ABB RAPID module: SERVER.mod

MODULE SERVER
!
!  Released under MIT License
!
!  David Pollard
!  Bristol Robotics Laboratory
!
!  Original author
!  Michael Dawson-Haggerty
!
!

!////////////////
!GLOBAL VARIABLES
!////////////////

! Robot configuration
PERS tooldata currentTool := [TRUE,[[-44.5,9.9,114],[1,0,0,0]],[0.001,[0,0,0.001],[1,0,0,0],0,0,0]];
PERS wobjdata currentWobj := [FALSE,TRUE,"",[[0,0,0],[1,0,0,0]],[[633.5,9.9,380],[1,0,0,0]]];
PERS speeddata currentSpeed;
PERS zonedata currentZone;

! Clock Synchronization
PERS bool startLog:=TRUE;
PERS bool startRob:=TRUE;

! Mutex between logger and changing the tool and work objects
PERS bool frameMutex:=FALSE;

! PC communication
VAR socketdev clientSocket;
VAR socketdev serverSocket;
VAR num instructionCode;
VAR num params{10};
VAR num nParams;

VAR num qOrientation{4};  !store Q value for orientation
VAR num tempNum;          !For use whenever needed. Don't rely on it to stay the same

!PERS string ipController:= "192.168.125.1"; !robot default IP
PERS string ipController:= "127.0.0.1"; !local IP for testing in simulation
PERS num serverPort:= 5000;

! Motion of the robot
VAR robtarget cartesianTarget;
VAR jointtarget jointsTarget;
VAR bool moveCompleted; !Set to true after finishing a Move instruction.

! Buffered move variables
CONST num MAX_BUFFER := 512;
CONST num MAX_SAVED_BUFFERS := 20;
VAR num BUFFER_POS := 0;
VAR robtarget bufferTargets{MAX_BUFFER};
VAR speeddata bufferSpeeds{MAX_BUFFER};
VAR bool extrudeDuringBufferMove;

! Spare buffers for saving paths
VAR robtarget savedBufferTargets{MAX_SAVED_BUFFERS, MAX_BUFFER};
VAR speeddata savedBufferSpeeds{MAX_SAVED_BUFFERS, MAX_BUFFER};
VAR num savedBufferPos{MAX_SAVED_BUFFERS};

! External axis position variables
VAR extjoint externalAxis;

! Circular move buffer
VAR robtarget circPoint;

! Correct Instruction Execution and possible return values
VAR num ok;
CONST num SERVER_BAD_MSG :=  0;
CONST num SERVER_OK := 1;
TASK PERS tooldata testNozzle:=[TRUE,[[-47.7913,12.961,103.954],[1,0,0,0]],[0.5,[0,0,0],[1,0,0,0],0,0,0]];
TASK PERS tooldata nozzle:=[TRUE,[[-44.5058,10.7853,113.761],[1,0,0,0]],[1,[0,0,0],[1,0,0,0],0,0,0]];


!////////////////
!LOCAL METHODS
!////////////////

! Method to parse the message received from a PC
!  If correct message, loads values on:
!  - instructionCode.
!  - nParams: Number of received parameters.
!  - params{nParams}: Vector of received params.
PROC ParseMsg(string msg)
    !//Local variables
    VAR bool auxOk;
    VAR num ind:=1;
    VAR num newInd;
    VAR num length;
    VAR num indParam:=1;
    VAR string subString;
    VAR bool end := FALSE;

    ! Find the end character
    length := StrMatch(msg,1,"#");
    IF length > StrLen(msg) THEN
        ! Corrupt message
        nParams := -1;
    ELSE
        ! Read Instruction code
        newInd := StrMatch(msg,ind," ") + 1;
        subString := StrPart(msg,ind,newInd - ind - 1);
        auxOk:= StrToVal(subString, instructionCode);
        IF auxOk = FALSE THEN
            ! Impossible to read instruction code
            nParams := -1;
        ELSE
            ind := newInd;
            ! Read all instruction parameters (maximum of 8)
            WHILE end = FALSE DO
                newInd := StrMatch(msg,ind," ") + 1;
                IF newInd > length THEN
                    end := TRUE;
                ELSE
                    subString := StrPart(msg,ind,newInd - ind - 1);
                    auxOk := StrToVal(subString, params{indParam});
                    indParam := indParam + 1;
                    ind := newInd;
                ENDIF
            ENDWHILE
            nParams:= indParam - 1;
        ENDIF
    ENDIF
ENDPROC


! Handshake between server and client:
!  - Creates socket.
!  - Waits for incoming TCP connection.
PROC ServerCreateAndConnect(string ip, num port)
    VAR string clientIP;

    SocketCreate serverSocket;
    SocketBind serverSocket, ip, port;
    SocketListen serverSocket;
    TPWrite "SERVER: Server waiting for incoming connections ...";
    WHILE SocketGetStatus(clientSocket) <> SOCKET_CONNECTED DO
        SocketAccept serverSocket,clientSocket \ClientAddress:=clientIP \Time:=WAIT_MAX;
        IF SocketGetStatus(clientSocket) <> SOCKET_CONNECTED THEN
            TPWrite "SERVER: Problem serving an incoming connection.";
            TPWrite "SERVER: Try reconnecting.";
        ENDIF
        ! Wait 0.5 seconds for the next reconnection
        WaitTime 0.5;
    ENDWHILE
    TPWrite "SERVER: Connected to IP " + clientIP;
ENDPROC


! Parameter initialization
!  Loads default values for
!  - Tool.
!  - WorkObject.
!  - Zone.
!  - Speed.
PROC Initialize()
    currentTool := [TRUE,[[0,0,0],[1,0,0,0]],[0.001,[0,0,0.001],[1,0,0,0],0,0,0]];
    currentWobj := [FALSE,TRUE,"",[[0,0,0],[1,0,0,0]],[[0,0,0],[1,0,0,0]]];
    currentSpeed := [100, 50, 0, 0];
    currentZone := [FALSE, 0.3, 0.3,0.3,0.03,0.3,0.03]; !z0

	!Find the current external axis values so they don't move when we start
    ActUnit STN1;
	jointsTarget := CJointT();
	externalAxis := jointsTarget.extax;
ENDPROC


!////////////////////////
!//SERVER: Main procedure
!////////////////////////
PROC ServerMain()
    ! Local variables
    VAR string receivedString;   ! Received string
    VAR string sendString;       ! Reply string
    VAR string addString;        ! String to add to the reply.
    VAR bool connected;          ! Client connected
    VAR bool reconnected;        ! Drop and reconnection happened during serving a command
    VAR robtarget cartesianPose;
    VAR jointtarget jointsPose;

    ! Motion configuration
    ConfL \Off;
    SingArea \Wrist;
    moveCompleted:= TRUE;

    ! Initialization of WorkObject, Tool, Speed and Zone
    Initialize;

    ! Socket connection
    connected:=FALSE;
    ServerCreateAndConnect ipController,serverPort;
    connected:=TRUE;

    ! Server Loop
    WHILE TRUE DO
        ! Initialization of program flow variables
        ok:=SERVER_OK;              ! Correctness of executed instruction.
        reconnected:=FALSE;         ! Has communication dropped after receiving a command?
        addString := "";

        ! Wait for a command
        SocketReceive clientSocket \Str:=receivedString \Time:=WAIT_MAX;
        ParseMsg receivedString;

        ! Execution of the command
        TEST instructionCode
            CASE -1:
                IF nParams = 1 THEN
                    IF params{1} = -1 THEN
                        ChangeExtruderState (0);
                        DeactUnit STN1;
                    ELSEIF params{1} = 0 THEN
                        ResetRobotPosition;
                        ChangeExtruderState(0);
                        DeactUnit STN1;
                    ELSEIF params{1} = 1 THEN
                        ResetRobotPosition;
                        ChangeExtruderState(1);
                        ActUnit STN1;
                    ELSEIF params{1} = 2 THEN
                        ChangeExtruderState(1);
                        ActUnit STN1;
                    ENDIF
                    ok := SERVER_OK;
                ELSE
                    ok := SERVER_BAD_MSG;
                ENDIF


            CASE 0: !Ping
                IF nParams = 0 THEN
                    ok := SERVER_OK;
                ELSE
                    ok := SERVER_BAD_MSG;
                ENDIF

            CASE 1: !Cartesian Move
                IF nParams = 8 THEN
                    jointsTarget := CJointT();
	                externalAxis := jointsTarget.extax;

                    cartesianTarget :=[[params{2},params{3},params{4}],
                                       [params{5},params{6},params{7},params{8}],
                                       [0,0,0,0],
                                       externalAxis];
                    ok := SERVER_OK;
                    moveCompleted := FALSE;
                    IF params{1}=1 THEN
                        MoveL cartesianTarget, currentSpeed, fine, currentTool \WObj:=currentWobj ;
                    ELSE
                        MoveL cartesianTarget, currentSpeed, currentZone, currentTool \WObj:=currentWobj ;
                    ENDIF
                    moveCompleted := TRUE;
                ELSE
                    ok := SERVER_BAD_MSG;
                ENDIF

            CASE 2: !Joint Move
                IF nParams = 6 THEN
                    jointsTarget := CJointT();
                    externalAxis := jointsTarget.extax;

                    jointsTarget:=[[params{1},params{2},params{3},params{4},params{5},params{6}], externalAxis];
                    ok := SERVER_OK;
                    moveCompleted := FALSE;
                    MoveAbsJ jointsTarget, currentSpeed, currentZone, currentTool \Wobj:=currentWobj;
                    moveCompleted := TRUE;
                ELSE
                    ok :=SERVER_BAD_MSG;
                ENDIF

            CASE 3: !Get Cartesian Coordinates (with current tool and workobject)
                IF nParams = 0 THEN
                    cartesianPose := CRobT(\Tool:=currentTool \WObj:=currentWObj);
                    addString := NumToStr(cartesianPose.trans.x,2) + " ";
                    addString := addString + NumToStr(cartesianPose.trans.y,2) + " ";
                    addString := addString + NumToStr(cartesianPose.trans.z,2) + " ";
                    addString := addString + NumToStr(cartesianPose.rot.q1,3) + " ";
                    addString := addString + NumToStr(cartesianPose.rot.q2,3) + " ";
                    addString := addString + NumToStr(cartesianPose.rot.q3,3) + " ";
                    addString := addString + NumToStr(cartesianPose.rot.q4,3); !End of string
                    ok := SERVER_OK;
                ELSE
                    ok :=SERVER_BAD_MSG;
                ENDIF

            CASE 4: !Get Joint Coordinates
                IF nParams = 0 THEN
                    jointsPose := CJointT();
                    addString := NumToStr(jointsPose.robax.rax_1,2) + " ";
                    addString := addString + NumToStr(jointsPose.robax.rax_2,2) + " ";
                    addString := addString + NumToStr(jointsPose.robax.rax_3,2) + " ";
                    addString := addString + NumToStr(jointsPose.robax.rax_4,2) + " ";
                    addString := addString + NumToStr(jointsPose.robax.rax_5,2) + " ";
                    addString := addString + NumToStr(jointsPose.robax.rax_6,2); !End of string
                    ok := SERVER_OK;
                ELSE
                    ok:=SERVER_BAD_MSG;
                ENDIF

			CASE 5: !Get external axis positions
                IF nParams=0 THEN
                    jointsTarget:=CJointT();
                    addString:=ValToStr(jointsTarget.extax.eax_b)+" ";
                    addString:=addString + ValToStr(jointsTarget.extax.eax_c);
                    ok:=SERVER_OK;
                ELSE
                    ok:=SERVER_BAD_MSG;
                ENDIF            CASE 6: !Set Tool
                IF nParams = 7 THEN
		            WHILE (frameMutex) DO
		                WaitTime .01; !  If the frame is being used by logger, wait here
		            ENDWHILE
		            frameMutex:= TRUE;
                    currentTool.tframe.trans.x:=params{1};
                    currentTool.tframe.trans.y:=params{2};
                    currentTool.tframe.trans.z:=params{3};
                    currentTool.tframe.rot.q1:=params{4};
                    currentTool.tframe.rot.q2:=params{5};
                    currentTool.tframe.rot.q3:=params{6};
                    currentTool.tframe.rot.q4:=params{7};
                    ok := SERVER_OK;
		            frameMutex:= FALSE;
                ELSE
                    ok:=SERVER_BAD_MSG;
                ENDIF

            CASE 7: !Set Work Object
                IF nParams = 7 THEN
                    currentWobj.oframe.trans.x:=params{1};
                    currentWobj.oframe.trans.y:=params{2};
                    currentWobj.oframe.trans.z:=params{3};
                    currentWobj.oframe.rot.q1:=params{4};
                    currentWobj.oframe.rot.q2:=params{5};
                    currentWobj.oframe.rot.q3:=params{6};
                    currentWobj.oframe.rot.q4:=params{7};
                    ok := SERVER_OK;
                ELSE
                    ok:=SERVER_BAD_MSG;
                ENDIF

            CASE 8: !Set Speed of the Robot
                IF nParams = 4 THEN
                    currentSpeed.v_tcp:=params{1};
                    currentSpeed.v_ori:=params{2};
                    currentSpeed.v_leax:=params{3};
                    currentSpeed.v_reax:=params{4};
                    ok := SERVER_OK;
                ELSEIF nParams = 2 THEN
					currentSpeed.v_tcp:=params{1};
					currentSpeed.v_ori:=params{2};
					ok := SERVER_OK;
				ELSE
                    ok:=SERVER_BAD_MSG;
                ENDIF

            CASE 9: !Set zone data
                IF nParams = 4 THEN
                    IF params{1}=1 THEN
                        currentZone.finep := TRUE;
                        currentZone.pzone_tcp := 0.0;
                        currentZone.pzone_ori := 0.0;
                        currentZone.zone_ori := 0.0;
                    ELSE
                        currentZone.finep := FALSE;
                        currentZone.pzone_tcp := params{2};
                        currentZone.pzone_ori := params{3};
                        currentZone.zone_ori := params{4};
                    ENDIF
                    ok := SERVER_OK;
                ELSE
                    ok:=SERVER_BAD_MSG;
                ENDIF

            CASE 10: !Rotate about tool Z axis
                IF nParams = 1 THEN
                    ok := SERVER_OK;
                    RotateToolZ(params{1});
                ELSE
                    ok := SERVER_BAD_MSG;
                ENDIF

            CASE 11: !Check and fix Joint 6 angle
                IF nParams = 0 THEN
                    ok := SERVER_OK;
                    jointsTarget := CJointT();
                    tempNum := jointsTarget.robax.rax_6;
                    ! Move and rotate if necessary
                    IF tempNum > 270 THEN
                        TPWrite "Performing angle correction";
                        cartesianPose := CRobT();
                        MoveL RelTool(cartesianPose,0,0,-50),v100,fine,currentTool \WObj:=currentWobj;
                        RotateToolZ(-360);
                        MoveL cartesianPose,v100,fine,currentTool \WObj:=currentWobj;
                    ELSEIF tempNum < -90 THEN
                        TPWrite "Performing angle correction";
                        cartesianPose := CRobT();
                        MoveL RelTool(cartesianPose,0,0,-50),v100,fine,currentTool \WObj:=currentWobj;
                        RotateToolZ(360);
                        MoveL cartesianPose,v100,fine,currentTool \WObj:=currentWobj;
                    ENDIF
                ELSE
                    ok := SERVER_BAD_MSG;
                ENDIF


            CASE 29:
                IF nParams = 4 THEN
                    qOrientation{1} := params{1};
                    qOrientation{2} := params{2};
                    qOrientation{3} := params{3};
                    qOrientation{4} := params{4};
                    ok:=SERVER_OK;
                ELSE
                    ok:=SERVER_BAD_MSG;
                ENDIF

            CASE 30: !Add Cartesian Coordinates to buffer
                IF nParams = 7 OR nParams = 8 THEN
                    ! If external axis is necessary
                    jointsTarget := CJointT();
                    externalAxis := jointsTarget.extax;
                    IF nParams = 8 THEN
                        externalAxis.eax_c := params{8};
                    ENDIF

                    cartesianTarget :=[[params{1},params{2},params{3}],
                                        [params{4},params{5},params{6},params{7}],
                                        [0,0,0,0],
                                        externalAxis];
                    IF BUFFER_POS < MAX_BUFFER THEN
                        BUFFER_POS := BUFFER_POS + 1;
                        bufferTargets{BUFFER_POS} := cartesianTarget;
                        bufferSpeeds{BUFFER_POS} := currentSpeed;
                    ENDIF
                    ! Update Q orienatation
                    qOrientation{1} := params{4};
                    qOrientation{2} := params{5};
                    qOrientation{3} := params{6};
                    qOrientation{4} := params{7};
                    ok := SERVER_OK;
                ELSEIF nParams = 3 THEN
                    cartesianTarget :=[[params{1},params{2},params{3}],
                                        [qOrientation{1},qOrientation{2},qOrientation{3},qOrientation{4}],
                                        [0,0,0,0],
                                        externalAxis];
                    IF BUFFER_POS < MAX_BUFFER THEN
                        BUFFER_POS := BUFFER_POS + 1;
                        bufferTargets{BUFFER_POS} := cartesianTarget;
                        bufferSpeeds{BUFFER_POS} := currentSpeed;
                    ENDIF
                    ok:=SERVER_OK;
                ELSE
                    ok:=SERVER_BAD_MSG;
                ENDIF

            CASE 31: !Clear Cartesian Buffer
                IF nParams = 0 THEN
                    BUFFER_POS := 0;
                    ok := SERVER_OK;
                ELSE
                    ok:=SERVER_BAD_MSG;
                ENDIF

            CASE 32: !Get Buffer Size)
                IF nParams = 0 THEN
                    addString := NumToStr(BUFFER_POS,2);
                    ok := SERVER_OK;
                ELSE
                    ok:=SERVER_BAD_MSG;
                ENDIF

            CASE 33: !Execute moves in cartesianBuffer as linear moves NB: Circ buffer is 37
                IF nParams = 0 OR nParams = 1 THEN
                    IF nParams = 1 THEN
                        MoveL bufferTargets{1}, v100, fine, currentTool, \WObj:=currentWobj ;
                        SetDO DO10_2, 1;
                        ! Ensure signal is synchronised
                        MoveL bufferTargets{1}, v100, fine, currentTool, \WObj:=currentWobj ;
                    ENDIF

                    FOR i FROM 1 TO (BUFFER_POS) DO
                        MoveL bufferTargets{i}, bufferSpeeds{i}, currentZone, currentTool, \WObj:=currentWobj ;
                    ENDFOR

                    MoveL bufferTargets{(BUFFER_POS)}, bufferSpeeds{(BUFFER_POS)}, fine, currentTool, \WObj:=currentWobj ;

                    IF nParams = 1 THEN
                        SetDO DO10_2, 0;
                        MoveL RelTool(bufferTargets{(BUFFER_POS)},0,0,-5),v100,z1, currentTool, \WObj:=currentWobj ;
                    ENDIF


                    ok := SERVER_OK;
                ELSE
                    ok:=SERVER_BAD_MSG;
                ENDIF

            CASE 34: !External Axis move
                IF nParams = 2 THEN
                    jointsTarget := CJointT();
                    jointsTarget.extax.eax_b := params{1};
                    jointsTarget.extax.eax_c := params{2};
                    ok := SERVER_OK;
                    moveCompleted := FALSE;
                    MoveAbsJ jointsTarget, currentSpeed, fine, currentTool \Wobj:=currentWobj;
                    moveCompleted := TRUE;
                ELSE
                    ok :=SERVER_BAD_MSG;
                ENDIF

            CASE 35: !Specify circPoint for circular move, and then wait on toPoint
                IF nParams = 7 THEN
                    jointsTarget := CJointT();
                    externalAxis := jointsTarget.extax;

                    circPoint :=[[params{1},params{2},params{3}],
                                [params{4},params{5},params{6},params{7}],
                                [0,0,0,0],
                                externalAxis];
                    TPWrite "z: ", \Num:=params{3};
                    ok := SERVER_OK;
                ELSE
                    ok:=SERVER_BAD_MSG;
                ENDIF

            CASE 36: !specify toPoint, and use circPoint specified previously
                IF nParams = 7 THEN
                    jointsTarget := CJointT();
                    externalAxis := jointsTarget.extax;

                    cartesianTarget :=[[params{1},params{2},params{3}],
                                        [params{4},params{5},params{6},params{7}],
                                        [0,0,0,0],
                                        externalAxis];
                    MoveC circPoint, cartesianTarget, currentSpeed, currentZone, currentTool \WObj:=currentWobj ;
                    ok := SERVER_OK;
                ELSE
                    ok:=SERVER_BAD_MSG;
                ENDIF

            CASE 37: !execute buffer as a circular move
                IF nParams = 0 THEN
                    MoveC bufferTargets{1}, bufferTargets{2}, bufferSpeeds{1}, currentZone, currentTool \WObj:=currentWobj ;
                    ok  := SERVER_OK;
                ELSE
                    ok := SERVER_BAD_MSG;
                ENDIF


            CASE 40:  ! Find if position is reachable
                ! NB: Not recommended for calling during operation, no error handling.
                cartesianTarget :=[[params{1},params{2},params{3}],
                                    [params{4},params{5},params{6},params{7}],
                                    [0,0,0,0],
                                    externalAxis];
                IF CheckPositionReachable(cartesianTarget, currentTool, currentWobj) THEN
                    ok := SERVER_OK;
                ELSE
                    ok := SERVER_BAD_MSG;
                ENDIF




            CASE 50: !Save current buffer into existing buffer
                IF nParams = 1 THEN
                    IF params{1} < MAX_SAVED_BUFFERS THEN
                        ok := SERVER_OK;
                        TPWrite "Saved: ",\Num:=params{1};
                        FOR i FROM 1 TO BUFFER_POS DO
                            savedBufferTargets{params{1},i} := bufferTargets{i};
                            savedBufferSpeeds{params{1},i} := bufferSpeeds{i};
                        ENDFOR
                        savedBufferPos{params{1}} := BUFFER_POS;
                    ELSE
                        ErrWrite "Buffer error", "Requested buffer does not exist";
                        ok := SERVER_BAD_MSG;
                    ENDIF
                ELSE
                    ok := SERVER_BAD_MSG;
                ENDIF

            CASE 51: !Load saved buffer into current buffer. Reset BUFFER_POS
                IF nParams=1 THEN
                    IF params{1} < MAX_SAVED_BUFFERS THEN
                        ok:=SERVER_OK;
                        BUFFER_POS := savedBufferPos{params{1}};
                        FOR i FROM 1 TO BUFFER_POS DO
                            bufferTargets{i} := savedBufferTargets{params{1},i};
                            bufferSpeeds{i} := savedBufferSpeeds{params{1},i};
                        ENDFOR
                    ELSE
                        ErrWrite "Buffer error", "Requested buffer does not exist";
                        ok := SERVER_BAD_MSG;
                    ENDIF
                ELSE
                    ok:=SERVER_BAD_MSG;
                ENDIF

            CASE 52: ! Read specific position from buffer
                IF nParams = 1 THEN
                    cartesianPose := bufferTargets{params{1}};
                    addString := NumToStr(cartesianPose.trans.x,2) + " ";
                    addString := addString + NumToStr(cartesianPose.trans.y,2) + " ";
                    addString := addString + NumToStr(cartesianPose.trans.z,2) + " ";
                    addString := addString + NumToStr(cartesianPose.rot.q1,3) + " ";
                    addString := addString + NumToStr(cartesianPose.rot.q2,3) + " ";
                    addString := addString + NumToStr(cartesianPose.rot.q3,3) + " ";
                    addString := addString + NumToStr(cartesianPose.rot.q4,3); !End of string
                    ok := SERVER_OK;

                    ok:= SERVER_OK;
                ELSE
                    ok := SERVER_BAD_MSG;
                ENDIF

            CASE 53: ! Offsets entire current buffer by set amount
                IF nParams = 3 THEN
                    ok := SERVER_OK;
                    FOR i FROM 1 TO BUFFER_POS DO
                        bufferTargets{i} := Offs(bufferTargets{i},params{1}, params{2}, params{3});
                    ENDFOR
                ELSE
                    ok := SERVER_BAD_MSG;
                ENDIF

            CASE 54:  ! Scale saved buffer speed
                IF nParams = 1 THEN
                    ok := SERVER_OK;
                    FOR i FROM 1 TO BUFFER_POS DO
                        bufferSpeeds{i}.v_tcp := bufferSpeeds{i}.v_tcp * params{1};
                    ENDFOR
                    TPWrite "Buffer speed multiplied by: " \Num:=params{1};
                ELSE
                    ok := SERVER_BAD_MSG;
                ENDIF


            CASE 97: ! Change DO port 2
                IF nParams = 1 THEN
                    IF params{1}=1 THEN
                        SetDO DO10_2, 1 ;
                    ELSE
                        SetDO DO10_2, 0 ;
                    ENDIF
                    ok :=SERVER_OK;
                ELSE
                    ok :=SERVER_BAD_MSG;
                ENDIF

            CASE 96: ! Set Group Output
                IF nParams = 1 THEN
                    TPWrite "Input: ", \Num:=params{1};
                    SetGO GO_Signal, params{1};
                    ok := SERVER_OK;
                ELSE
                    ok := SERVER_BAD_MSG;
                ENDIF

            CASE 98: !returns current robot info: serial number, robotware version, and robot type
                IF nParams = 0 THEN
                    addString := GetSysInfo(\SerialNo) + "*";
                    addString := addString + GetSysInfo(\SWVersion) + "*";
                    addString := addString + GetSysInfo(\RobotType);
                    ok := SERVER_OK;
                ELSE
                    ok :=SERVER_BAD_MSG;
                ENDIF

            CASE 99: !Close Connection
                IF nParams = 0 THEN
                    TPWrite "SERVER: Client has closed connection.";
                    connected := FALSE;
                    ! Closing the server
                    SocketClose clientSocket;
                    SocketClose serverSocket;

                    !Reinitiate the server
                    ServerCreateAndConnect ipController,serverPort;
                    connected := TRUE;
                    reconnected := TRUE;
                    ok := SERVER_OK;
                ELSE
                    ok := SERVER_BAD_MSG;
                ENDIF
            DEFAULT:
                TPWrite "SERVER: Illegal instruction code";
                ok := SERVER_BAD_MSG;
        ENDTEST

        !Compose the acknowledge string to send back to the client
        IF connected = TRUE THEN
            IF reconnected = FALSE THEN
			    IF SocketGetStatus(clientSocket) = SOCKET_CONNECTED THEN
				    sendString := NumToStr(instructionCode,0);
                    sendString := sendString + " " + NumToStr(ok,0);
                    sendString := sendString + " " + addString;
                    SocketSend clientSocket \Str:=sendString;
			    ENDIF
            ENDIF
        ENDIF
    ENDWHILE

ERROR (LONG_JMP_ALL_ERR)
    TPWrite "SERVER: ------";
    TPWrite "SERVER: Error Handler:" + NumtoStr(ERRNO,0);
    TEST ERRNO
        CASE ERR_SOCK_CLOSED:
            TPWrite "SERVER: Lost connection to the client.";
            TPWrite "SERVER: Closing socket and restarting.";
            TPWrite "SERVER: ------";
            connected:=FALSE;
            ! Closing the server
            SocketClose clientSocket;
            SocketClose serverSocket;
            ! Reinitiate the server
            ServerCreateAndConnect ipController,serverPort;
            reconnected:= FALSE;
            connected:= TRUE;
            RETRY;
        DEFAULT:
            TPWrite "SERVER: Unknown error.";
            TPWrite "SERVER: Closing socket and restarting.";
            TPWrite "SERVER: ------";
            connected:=FALSE;
            ! Closing the server
            SocketClose clientSocket;
            SocketClose serverSocket;
            ! Reinitiate the server
            ServerCreateAndConnect ipController,serverPort;
            reconnected:= FALSE;
            connected:= TRUE;
            RETRY;
    ENDTEST
ENDPROC

PROC ResetRobotPosition()
    VAR jointtarget HomePose;
    VAR robtarget pTemp;
    ActUnit STN1;
    pTemp := CRobT();
    pTemp.extax.eax_b := 0;
    pTemp.extax.eax_c := 0;
    HomePose := [[0,0,0,0,0,0], pTemp.extax];
    SetDO DO10_1, 0;
    SetDO DO10_2, 0;
    SetDO DO10_3, 0;
    SetDO DO10_4, 0;
    SetDO DO10_5, 0;
    SetDO DO10_6, 0;
    SetDO DO10_7, 0;
    SetDO DO10_8, 0;
    SetDO DO10_9, 0;
    SetDO DO10_10, 0;
    SetDO DO10_11, 0;
    SetDO DO10_12, 0;
    MoveAbsJ HomePose, v200, fine, tool0;
    DeactUnit STN1;
    TPWrite "Reset complete";
ENDPROC

PROC RotateToolZ(num reqAngle)
    VAR robtarget tempPose;
    VAR num numRotations;
    tempPose := CRobT();
    numRotations := 0;
    WHILE Abs(reqAngle) > 45 DO
        numRotations := numRotations+1;
        IF reqAngle > 45 THEN
            MoveL RelTool(tempPose,0,0,0,\Rz:=numRotations * 45),currentSpeed, z0, currentTool \Wobj:=currentWobj;
            reqAngle := reqAngle-45;
        ELSEIF reqAngle < -45 THEN
            MoveL RelTool(tempPose,0,0,0,\Rz:=-1 * numRotations * 45),currentSpeed, z0, currentTool \Wobj:=currentWobj;
            reqAngle := reqAngle+45;
        ENDIF
    ENDWHILE
    IF reqAngle>0 THEN
        numRotations := numRotations * 45 + reqAngle;
        MoveL RelTool(tempPose,0,0,0,\Rz:=numRotations),currentSpeed, fine, currentTool \Wobj:=currentWobj;
    ELSE
        numRotations := -1 * numRotations * 45 + reqAngle;
        MoveL RelTool(tempPose,0,0,0,\Rz:=numRotations),currentSpeed, fine, currentTool \Wobj:=currentWobj;
    ENDIF
ENDPROC

PROC ChangeExtruderState(num State) ! Pass 1 for enable extruder, anything else for disable
    IF State = 1 THEN
        SetDO DO10_1, 1;
    ELSE
        SetDO DO10_1, 0;
    ENDIF
ENDPROC

FUNC bool CheckPositionReachable(robtarget pTarget, PERS tooldata cTool, PERS wobjdata cWobj)
    VAR jointtarget testJointT;
    VAR bool bReturnVal := TRUE;
    testJointT := CalcJointT(pTarget, cTool \WObj:=cWobj);
    RETURN bReturnVal;
ERROR
    IF ERRNO=ERR_ROBLIMIT THEN
        SkipWarn;
        bReturnVal := FALSE;
        TRYNEXT;
    ENDIF
ENDFUNC

ENDMODULE
